FUNCTION F_GET_INT_IN_RANGE : INT
VAR_INPUT
	value, range_max, range_min, value_max, value_min : INT; // Where range max/min is the range you want to fit the value
END_VAR
VAR
END_VAR

F_GET_INT_IN_RANGE := ((LIMIT(value_min, value, value_max) - value_min)*(range_max - range_min))/(value_max-value_min) + range_min;

END_FUNCTION

(* stored: Version 1.1.0.1, ProductVersion 3.1.4024.9
   POU F_GET_INT_IN_RANGE: Id {1b0b04bb-1af9-4b9d-a0ec-f97d90bbf3aa}, SpecialFunc None *)
